(* IEC 61131-3 sources: CodesysTest/alpha/export/Device.dev/Plc Logic/Application/ObjectHandling/FB_CollectionHandlerInitializable.pou, 1 file *)

(* ---- FB_CollectionHandlerInitializable.pou.st ---- *)
(*#-#-#-#-#-#-#-#-#-#---Declaration---#-#-#-#-#-#-#-#-#-#-#-#-#*)

FUNCTION_BLOCK FB_CollectionHandlerInitializable
VAR_INPUT

END_VAR
VAR
	Collection: ARRAY[0..GlobalObjects.MAX_LOGGABLE] OF IInitializable; // object array
	ObjNames   : ARRAY[0..GlobalObjects.MAX_LOGGABLE] OF STRING;
	_ArrayOver   : BOOL;
	_BadObj      : INT;
	_DupeObj   : INT;
	_OverObj   : INT;
	_TotalObj   : UINT;
END_VAR(*#-#-#-#-#-#-#-#-#-#---Implementation---#-#-#-#-#-#-#-#-#-#-#-#-#*)

//	Function Block: FB_CollectionHandlerLoggable
//	Description: This collection handler takes in loggable objects and registers them with a logger.  The FirstScan function should trigger the
//				 RegisterAll() method to register all loggable objects with a logger
//	Created by: Ben Hess
//	Created Date: Tuesday, September 11, 2018
